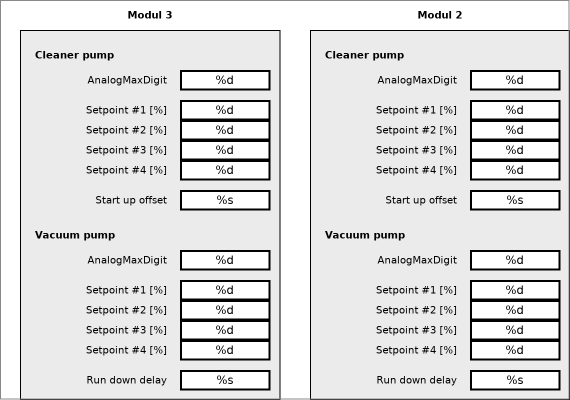
VISUALIZATION VISU_CLEAN_SEQUENCE  // 570x400
    Rectangle (20,30 260x370)
    Rectangle (180,70 90x20), "%d", text variable: PRG_MACHINE.fb_CleaningValvePump[2].lR_AnalogMaxDigitCleanerPump
        OnMouseDown: write the text variable via Default
    Rectangle (30,70 140x20), "AnalogMaxDigit"
    Rectangle (32,45 131x20), "Cleaner pump"
    Rectangle (180,100 90x20), "%d", text variable: PRG_MACHINE.fb_CleaningValvePump[2].lR_SetPoint1CleanerPump
        OnMouseDown: write the text variable via Default, min 0, max 100
    Rectangle (30,100 140x20), "Setpoint #1 [%]"
    Rectangle (180,120 90x20), "%d", text variable: PRG_MACHINE.fb_CleaningValvePump[2].lR_SetPoint2CleanerPump
        OnMouseDown: write the text variable via Default, min 0, max 100
    Rectangle (30,120 140x20), "Setpoint #2 [%]"
    Rectangle (180,140 90x20), "%d", text variable: PRG_MACHINE.fb_CleaningValvePump[2].lR_SetPoint3CleanerPump
        OnMouseDown: write the text variable via Default, min 0, max 100
    Rectangle (30,140 140x20), "Setpoint #3 [%]"
    Rectangle (180,160 90x20), "%d", text variable: PRG_MACHINE.fb_CleaningValvePump[2].lR_SetPoint4CleanerPump
        OnMouseDown: write the text variable via Default, min 0, max 100
    Rectangle (30,160 140x20), "Setpoint #4 [%]"
    Rectangle (180,250 90x20), "%d", text variable: PRG_MACHINE.fb_CleaningValvePump[2].lR_AnalogMaxDigitVacuumPump
        OnMouseDown: write the text variable via Default
    Rectangle (30,250 140x20), "AnalogMaxDigit"
    Rectangle (32,225 131x20), "Vacuum pump"
    Rectangle (180,280 90x20), "%d", text variable: PRG_MACHINE.fb_CleaningValvePump[2].lR_SetPoint1VacuumPump
        OnMouseDown: write the text variable via Default, min 0, max 100
    Rectangle (30,280 140x20), "Setpoint #1 [%]"
    Rectangle (180,300 90x20), "%d", text variable: PRG_MACHINE.fb_CleaningValvePump[2].lR_SetPoint2VacuumPump
        OnMouseDown: write the text variable via Default, min 0, max 100
    Rectangle (30,300 140x20), "Setpoint #2 [%]"
    Rectangle (180,320 90x20), "%d", text variable: PRG_MACHINE.fb_CleaningValvePump[2].lR_SetPoint3VacuumPump
        OnMouseDown: write the text variable via Default, min 0, max 100
    Rectangle (30,320 140x20), "Setpoint #3 [%]"
    Rectangle (180,340 90x20), "%d", text variable: PRG_MACHINE.fb_CleaningValvePump[2].lR_SetPoint4VacuumPump
        OnMouseDown: write the text variable via Default, min 0, max 100
    Rectangle (30,340 140x20), "Setpoint #4 [%]"
    Rectangle (180,190 90x20), "%s", text variable: PRG_MACHINE.fb_CleaningValvePump[2].tR_CleanerPumpOffset
        OnMouseDown: write the text variable via Default
    Rectangle (30,190 140x20), "Start up offset"
    Rectangle (180,370 90x20), "%s", text variable: PRG_MACHINE.fb_CleaningValvePump[2].tR_VacuumPumpDelay
        OnMouseDown: write the text variable via Default
    Rectangle (30,370 140x20), "Run down delay"
    Rectangle (310,30 260x370)
    Rectangle (470,70 90x20), "%d", text variable: PRG_MACHINE.fb_CleaningValvePump[1].lR_AnalogMaxDigitCleanerPump
        OnMouseDown: write the text variable via Default
    Rectangle (320,70 140x20), "AnalogMaxDigit"
    Rectangle (322,45 131x20), "Cleaner pump"
    Rectangle (470,100 90x20), "%d", text variable: PRG_MACHINE.fb_CleaningValvePump[1].lR_SetPoint1CleanerPump
        OnMouseDown: write the text variable via Default, min 0, max 100
    Rectangle (320,100 140x20), "Setpoint #1 [%]"
    Rectangle (470,120 90x20), "%d", text variable: PRG_MACHINE.fb_CleaningValvePump[1].lR_SetPoint2CleanerPump
        OnMouseDown: write the text variable via Default, min 0, max 100
    Rectangle (320,120 140x20), "Setpoint #2 [%]"
    Rectangle (470,140 90x20), "%d", text variable: PRG_MACHINE.fb_CleaningValvePump[1].lR_SetPoint3CleanerPump
        OnMouseDown: write the text variable via Default, min 0, max 100
    Rectangle (320,140 140x20), "Setpoint #3 [%]"
    Rectangle (470,160 90x20), "%d", text variable: PRG_MACHINE.fb_CleaningValvePump[1].lR_SetPoint4CleanerPump
        OnMouseDown: write the text variable via Default, min 0, max 100
    Rectangle (320,160 140x20), "Setpoint #4 [%]"
    Rectangle (470,250 90x20), "%d", text variable: PRG_MACHINE.fb_CleaningValvePump[1].lR_AnalogMaxDigitVacuumPump
        OnMouseDown: write the text variable via Default
    Rectangle (320,250 140x20), "AnalogMaxDigit"
    Rectangle (322,225 131x20), "Vacuum pump"
    Rectangle (470,280 90x20), "%d", text variable: PRG_MACHINE.fb_CleaningValvePump[1].lR_SetPoint1VacuumPump
        OnMouseDown: write the text variable via Default, min 0, max 100
    Rectangle (320,280 140x20), "Setpoint #1 [%]"
    Rectangle (470,300 90x20), "%d", text variable: PRG_MACHINE.fb_CleaningValvePump[1].lR_SetPoint2VacuumPump
        OnMouseDown: write the text variable via Default, min 0, max 100
    Rectangle (320,300 140x20), "Setpoint #2 [%]"
    Rectangle (470,320 90x20), "%d", text variable: PRG_MACHINE.fb_CleaningValvePump[1].lR_SetPoint3VacuumPump
        OnMouseDown: write the text variable via Default, min 0, max 100
    Rectangle (320,320 140x20), "Setpoint #3 [%]"
    Rectangle (470,340 90x20), "%d", text variable: PRG_MACHINE.fb_CleaningValvePump[1].lR_SetPoint4VacuumPump
        OnMouseDown: write the text variable via Default, min 0, max 100
    Rectangle (320,340 140x20), "Setpoint #4 [%]"
    Rectangle (470,190 90x20), "%s", text variable: PRG_MACHINE.fb_CleaningValvePump[1].tR_CleanerPumpOffset
        OnMouseDown: write the text variable via Default
    Rectangle (320,190 140x20), "Start up offset"
    Rectangle (470,370 90x20), "%s", text variable: PRG_MACHINE.fb_CleaningValvePump[1].tR_VacuumPumpDelay
        OnMouseDown: write the text variable via Default
    Rectangle (320,370 140x20), "Run down delay"
    Rectangle (310,5 260x20), "Modul 2"
    Rectangle (20,5 260x20), "Modul 3"
END_VISUALIZATION

(* stored: Version 1.1.0.1, ProductVersion 3.1.4024.9
   Visu VISU_CLEAN_SEQUENCE: Id {f4f504eb-ec61-4aa4-874b-ceb07b79bf59} *)
